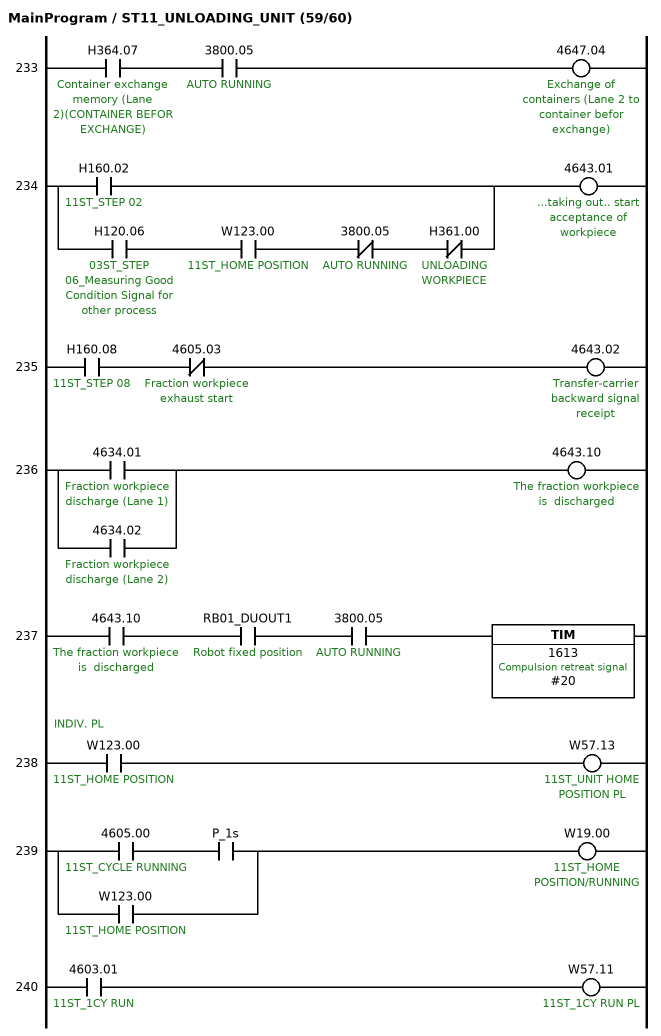
; [picture p576: MainProgram / ST11_UNLOADING_UNIT, rungs 233-240]
; rung 233
LD H364.07  ; Container exchange memory (Lane 2)(CONTAINER BEFOR EXCHANGE)
AND 3800.05  ; AUTO RUNNING
OUT 4647.04  ; Exchange of containers (Lane 2 to container befor exchange)
; rung 234
LD H160.02  ; 11ST_STEP 02
LD H120.06  ; 03ST_STEP 06_Measuring Good Condition Signal for other process
AND W123.00  ; 11ST_HOME POSITION
ANDNOT 3800.05  ; AUTO RUNNING
ANDNOT H361.00  ; UNLOADING WORKPIECE
ORLD
OUT 4643.01  ; ...taking out.. start acceptance of workpiece
; rung 235
LD H160.08  ; 11ST_STEP 08
ANDNOT 4605.03  ; Fraction workpiece exhaust start
OUT 4643.02  ; Transfer-carrier backward signal receipt
; rung 236
LD 4634.01  ; Fraction workpiece discharge (Lane 1)
OR 4634.02  ; Fraction workpiece discharge (Lane 2)
OUT 4643.10  ; The fraction workpiece is  discharged
; rung 237
LD 4643.10  ; The fraction workpiece is  discharged
AND RB01_DUOUT1  ; Robot fixed position
AND 3800.05  ; AUTO RUNNING
TIM 1613 #20  ; Compulsion retreat signal
; rung 238: INDIV. PL
LD W123.00  ; 11ST_HOME POSITION
OUT W57.13  ; 11ST_UNIT HOME POSITION PL
; rung 239
LD 4605.00  ; 11ST_CYCLE RUNNING
AND P_1s
OR W123.00  ; 11ST_HOME POSITION
OUT W19.00  ; 11ST_HOME POSITION/RUNNING
; rung 240
LD 4603.01  ; 11ST_1CY RUN
OUT W57.11  ; 11ST_1CY RUN PL

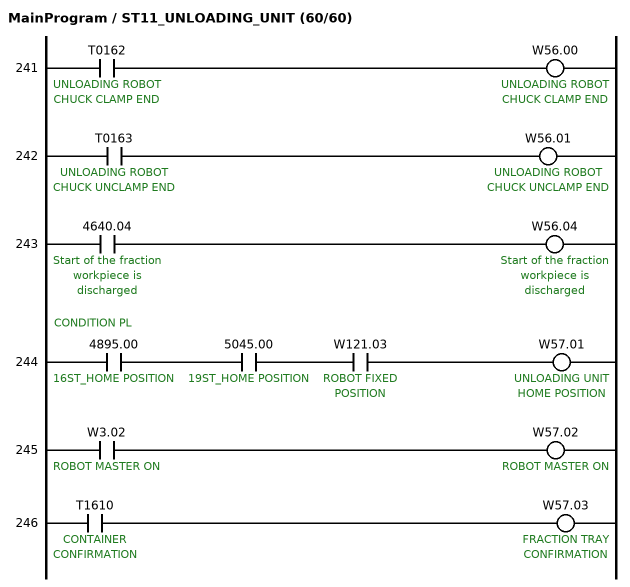
; rung 241
LD T0162  ; UNLOADING ROBOT CHUCK CLAMP END
OUT W56.00  ; UNLOADING ROBOT CHUCK CLAMP END
; rung 242
LD T0163  ; UNLOADING ROBOT CHUCK UNCLAMP END
OUT W56.01  ; UNLOADING ROBOT CHUCK UNCLAMP END
; rung 243
LD 4640.04  ; Start of the fraction workpiece is discharged
OUT W56.04  ; Start of the fraction workpiece is discharged
; rung 244: CONDITION PL
LD 4895.00  ; 16ST_HOME POSITION
AND 5045.00  ; 19ST_HOME POSITION
AND W121.03  ; ROBOT FIXED POSITION
OUT W57.01  ; UNLOADING UNIT HOME POSITION
; rung 245
LD W3.02  ; ROBOT MASTER ON
OUT W57.02  ; ROBOT MASTER ON
; rung 246
LD T1610  ; CONTAINER CONFIRMATION
OUT W57.03  ; FRACTION TRAY CONFIRMATION

### Section ST12_BEARING_SUPPLY_UNIT
; rung 0: 12ST_BEARING SUPPLY UNIT

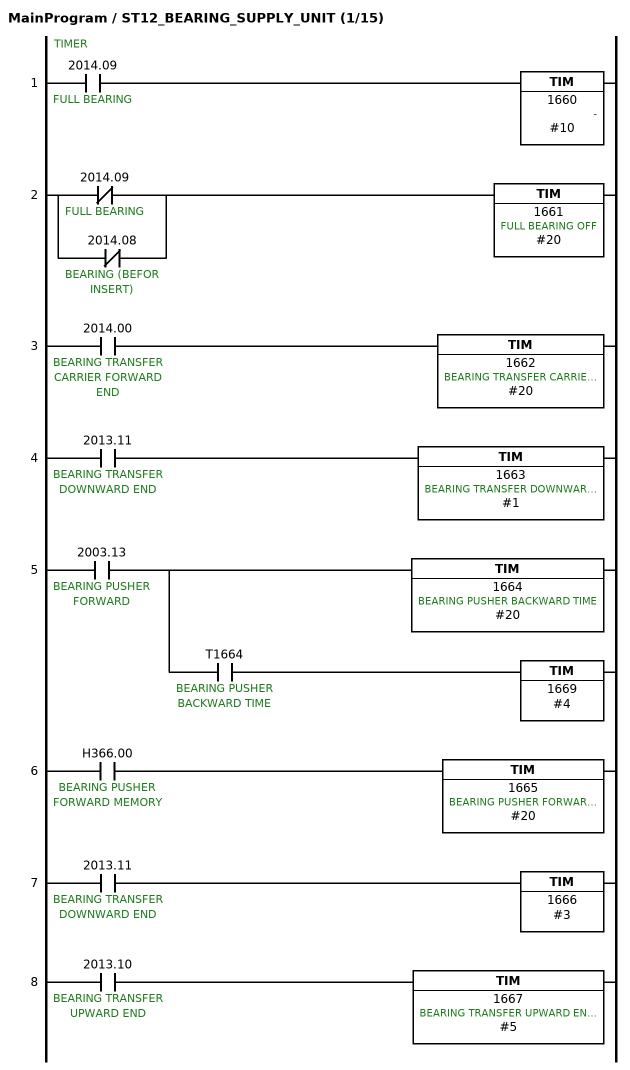
; rung 1: TIMER
LD 2014.09  ; FULL BEARING
TIM 1660 #10  ; -
; rung 2
LDNOT 2014.09  ; FULL BEARING
ORNOT 2014.08  ; BEARING (BEFOR INSERT)
TIM 1661 #20  ; FULL BEARING OFF
; rung 3
LD 2014.00  ; BEARING TRANSFER CARRIER FORWARD END
TIM 1662 #20  ; BEARING TRANSFER CARRIER FORWARD END TIME
; rung 4
LD 2013.11  ; BEARING TRANSFER DOWNWARD END
TIM 1663 #1  ; BEARING TRANSFER DOWNWARD END TIME
; rung 5
LD 2003.13  ; BEARING PUSHER FORWARD
TIM 1664 #20  ; BEARING PUSHER BACKWARD TIME
AND T1664  ; BEARING PUSHER BACKWARD TIME
TIM 1669 #4
; rung 6
LD H366.00  ; BEARING PUSHER FORWARD MEMORY
TIM 1665 #20  ; BEARING PUSHER FORWARD MEMORY TIME
; rung 7
LD 2013.11  ; BEARING TRANSFER DOWNWARD END
TIM 1666 #3
; rung 8
LD 2013.10  ; BEARING TRANSFER UPWARD END
TIM 1667 #5  ; BEARING TRANSFER UPWARD END CONFIRMATION

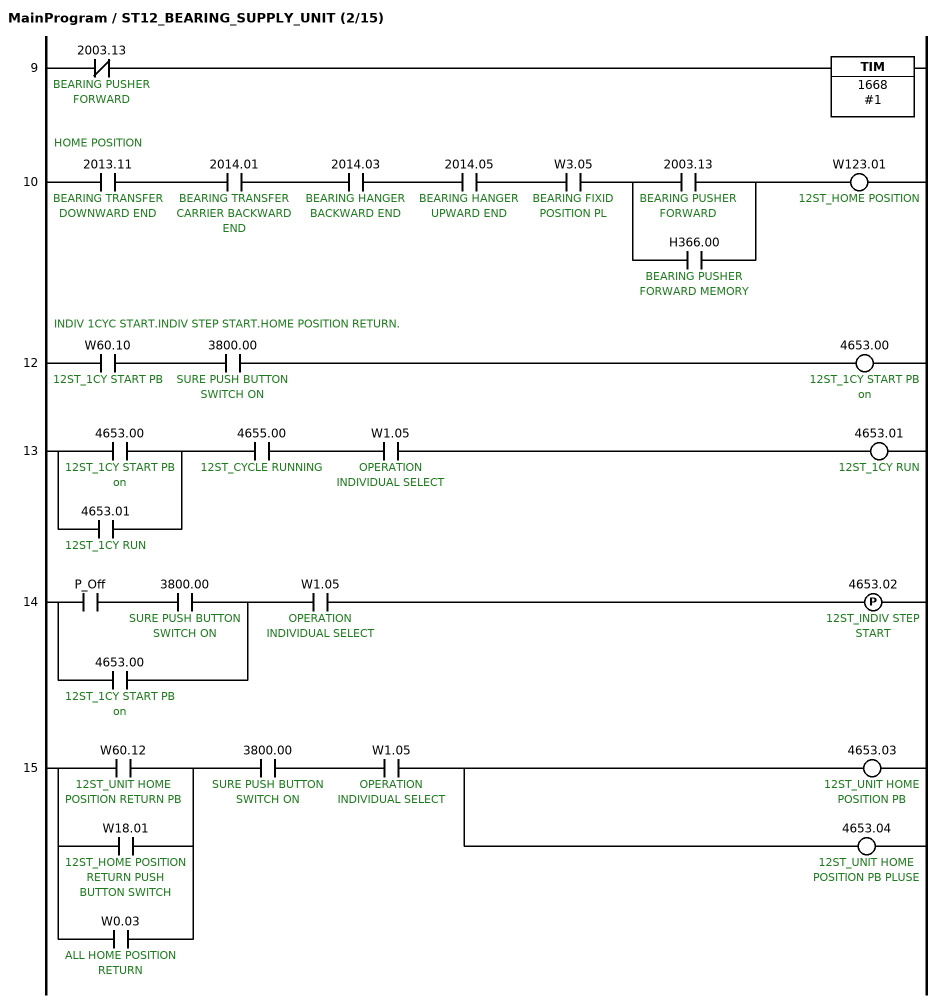
; rung 9
LDNOT 2003.13  ; BEARING PUSHER FORWARD
TIM 1668 #1
; rung 10: HOME POSITION
LD 2013.11  ; BEARING TRANSFER DOWNWARD END
AND 2014.01  ; BEARING TRANSFER CARRIER BACKWARD END
AND 2014.03  ; BEARING HANGER BACKWARD END
AND 2014.05  ; BEARING HANGER UPWARD END
AND W3.05  ; BEARING FIXID POSITION PL
LD 2003.13  ; BEARING PUSHER FORWARD
OR H366.00  ; BEARING PUSHER FORWARD MEMORY
ANDLD
OUT W123.01  ; 12ST_HOME POSITION
; rung 11: INTERFERENCE
; rung 12: INDIV 1CYC START.INDIV STEP START.HOME POSITION RETURN.
LD W60.10  ; 12ST_1CY START PB
AND 3800.00  ; SURE PUSH BUTTON SWITCH ON
OUT 4653.00  ; 12ST_1CY START PB on
; rung 13
LD 4653.00  ; 12ST_1CY START PB on
OR 4653.01  ; 12ST_1CY RUN
AND 4655.00  ; 12ST_CYCLE RUNNING
AND W1.05  ; OPERATION INDIVIDUAL SELECT
OUT 4653.01  ; 12ST_1CY RUN
; rung 14
LD P_Off
AND 3800.00  ; SURE PUSH BUTTON SWITCH ON
OR 4653.00  ; 12ST_1CY START PB on
AND W1.05  ; OPERATION INDIVIDUAL SELECT
DIFU(013) 4653.02  ; 12ST_INDIV STEP START
; rung 15
LD W60.12  ; 12ST_UNIT HOME POSITION RETURN PB
OR W18.01  ; 12ST_HOME POSITION RETURN PUSH BUTTON SWITCH
OR W0.03  ; ALL HOME POSITION RETURN
AND 3800.00  ; SURE PUSH BUTTON SWITCH ON
AND W1.05  ; OPERATION INDIVIDUAL SELECT
OUT 4653.03  ; 12ST_UNIT HOME POSITION PB
OUT 4653.04  ; 12ST_UNIT HOME POSITION PB PLUSE

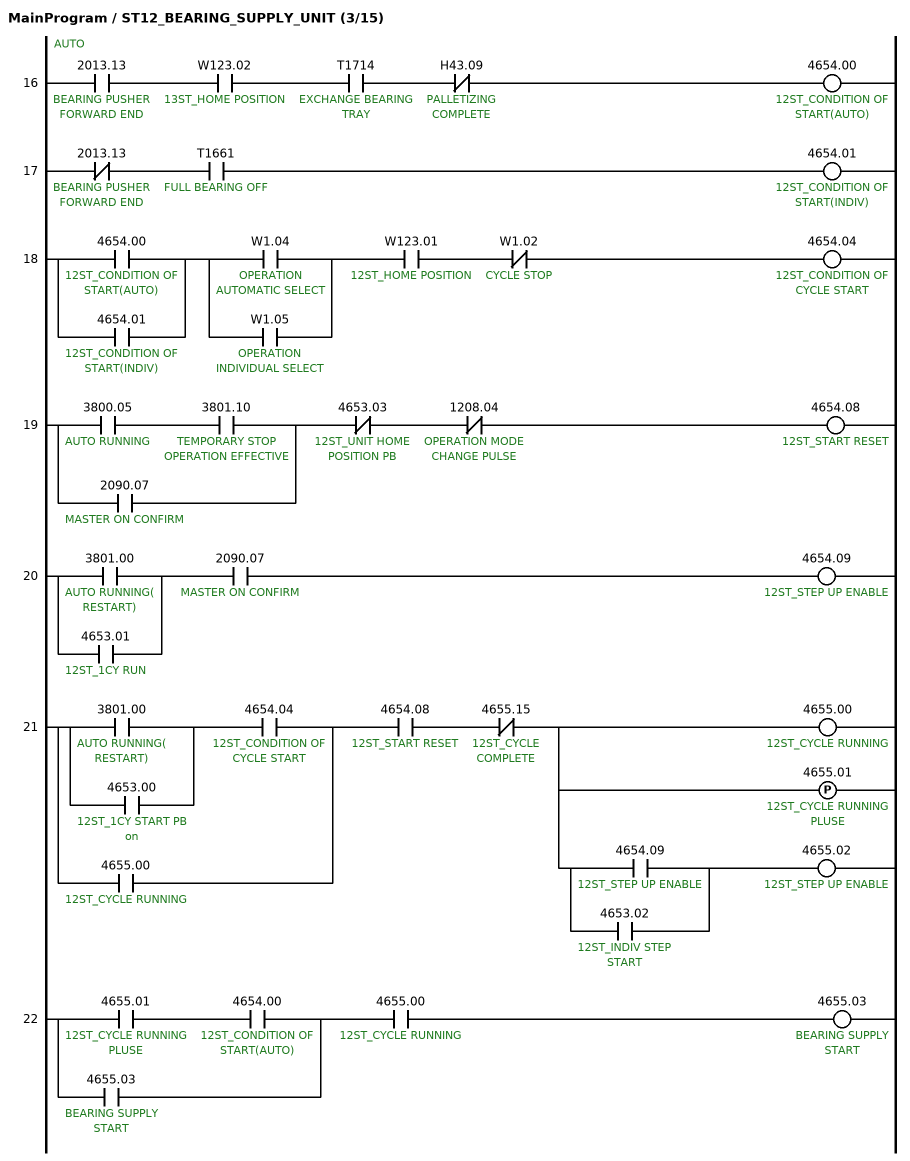
; rung 16: AUTO
LD 2013.13  ; BEARING PUSHER FORWARD END
AND W123.02  ; 13ST_HOME POSITION
AND T1714  ; EXCHANGE BEARING TRAY
ANDNOT H43.09  ; PALLETIZING COMPLETE
OUT 4654.00  ; 12ST_CONDITION OF START(AUTO)
; rung 17
LDNOT 2013.13  ; BEARING PUSHER FORWARD END
AND T1661  ; FULL BEARING OFF
OUT 4654.01  ; 12ST_CONDITION OF START(INDIV)
; rung 18
LD 4654.00  ; 12ST_CONDITION OF START(AUTO)
OR 4654.01  ; 12ST_CONDITION OF START(INDIV)
LD W1.04  ; OPERATION AUTOMATIC SELECT
OR W1.05  ; OPERATION INDIVIDUAL SELECT
ANDLD
AND W123.01  ; 12ST_HOME POSITION
ANDNOT W1.02  ; CYCLE STOP
OUT 4654.04  ; 12ST_CONDITION OF CYCLE START
; rung 19
LD 3800.05  ; AUTO RUNNING
AND 3801.10  ; TEMPORARY STOP OPERATION EFFECTIVE
OR 2090.07  ; MASTER ON CONFIRM
ANDNOT 4653.03  ; 12ST_UNIT HOME POSITION PB
ANDNOT 1208.04  ; OPERATION MODE CHANGE PULSE
OUT 4654.08  ; 12ST_START RESET
; rung 20
LD 3801.00  ; AUTO RUNNING(RESTART)
OR 4653.01  ; 12ST_1CY RUN
AND 2090.07  ; MASTER ON CONFIRM
OUT 4654.09  ; 12ST_STEP UP ENABLE
; rung 21
LD 3801.00  ; AUTO RUNNING(RESTART)
OR 4653.00  ; 12ST_1CY START PB on
AND 4654.04  ; 12ST_CONDITION OF CYCLE START
OR 4655.00  ; 12ST_CYCLE RUNNING
AND 4654.08  ; 12ST_START RESET
ANDNOT 4655.15  ; 12ST_CYCLE COMPLETE
OUT 4655.00  ; 12ST_CYCLE RUNNING
DIFU(013) 4655.01  ; 12ST_CYCLE RUNNING PLUSE
LD 4654.09  ; 12ST_STEP UP ENABLE
OR 4653.02  ; 12ST_INDIV STEP START
ANDLD
OUT 4655.02  ; 12ST_STEP UP ENABLE
; rung 22
LD 4655.01  ; 12ST_CYCLE RUNNING PLUSE
AND 4654.00  ; 12ST_CONDITION OF START(AUTO)
OR 4655.03  ; BEARING SUPPLY START
AND 4655.00  ; 12ST_CYCLE RUNNING
OUT 4655.03  ; BEARING SUPPLY START

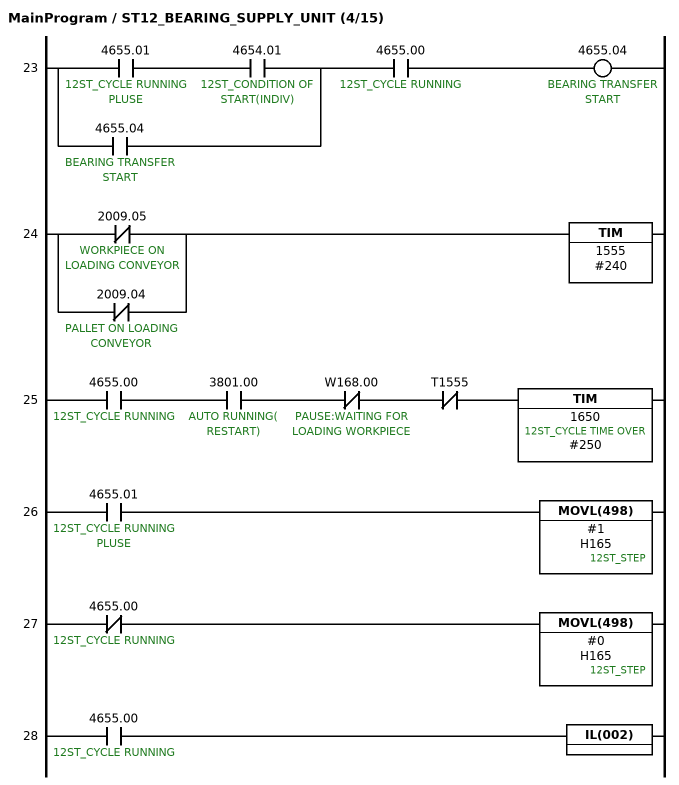
; rung 23
LD 4655.01  ; 12ST_CYCLE RUNNING PLUSE
AND 4654.01  ; 12ST_CONDITION OF START(INDIV)
OR 4655.04  ; BEARING TRANSFER START
AND 4655.00  ; 12ST_CYCLE RUNNING
OUT 4655.04  ; BEARING TRANSFER START
; rung 24
LDNOT 2009.05  ; WORKPIECE ON LOADING CONVEYOR
ORNOT 2009.04  ; PALLET ON LOADING CONVEYOR
TIM 1555 #240
; rung 25
LD 4655.00  ; 12ST_CYCLE RUNNING
AND 3801.00  ; AUTO RUNNING(RESTART)
ANDNOT W168.00  ; PAUSE:WAITING FOR LOADING WORKPIECE
ANDNOT T1555
TIM 1650 #250  ; 12ST_CYCLE TIME OVER
; rung 26
LD 4655.01  ; 12ST_CYCLE RUNNING PLUSE
MOVL(498) #1 H165  ; 12ST_STEP
; rung 27
LDNOT 4655.00  ; 12ST_CYCLE RUNNING
MOVL(498) #0 H165  ; 12ST_STEP
; rung 28
LD 4655.00  ; 12ST_CYCLE RUNNING
IL(002)

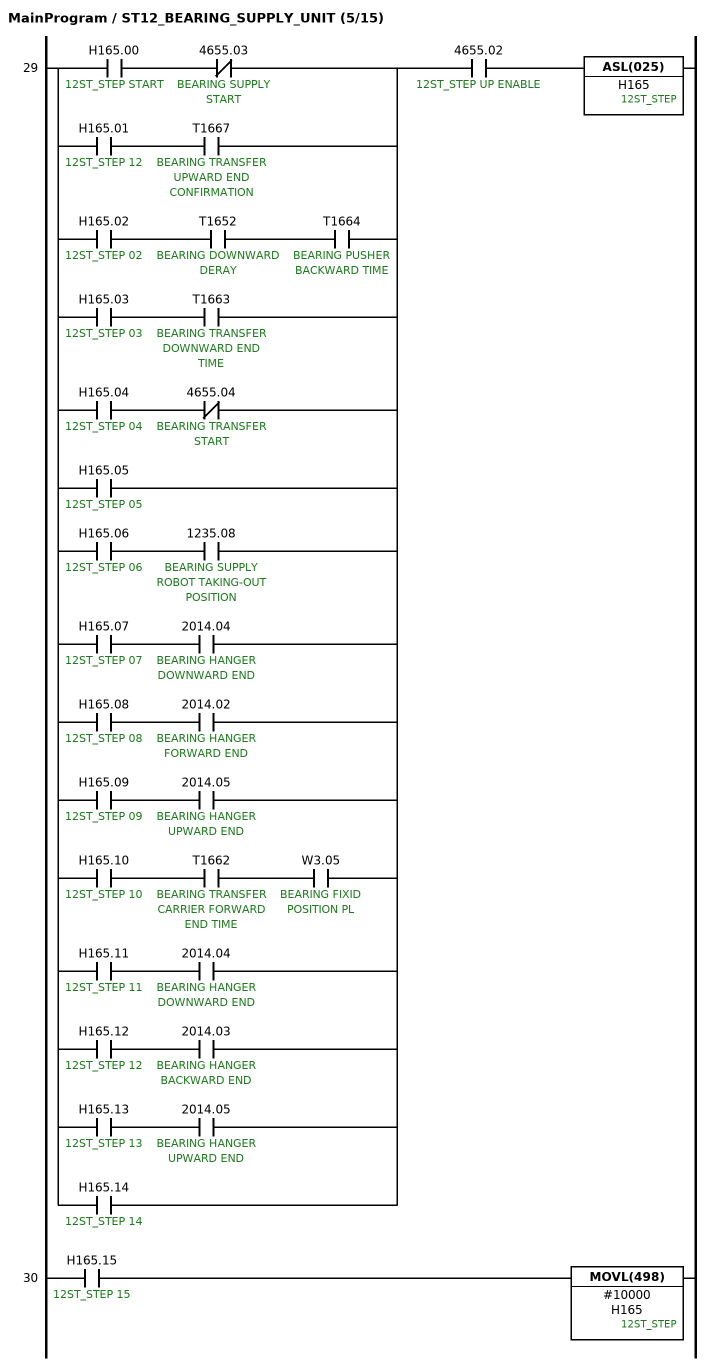
; rung 29
LD H165.00  ; 12ST_STEP START
ANDNOT 4655.03  ; BEARING SUPPLY START
LD H165.01  ; 12ST_STEP 12
AND T1667  ; BEARING TRANSFER UPWARD END CONFIRMATION
ORLD
LD H165.02  ; 12ST_STEP 02
AND T1652  ; BEARING DOWNWARD DERAY
AND T1664  ; BEARING PUSHER BACKWARD TIME
ORLD
LD H165.03  ; 12ST_STEP 03
AND T1663  ; BEARING TRANSFER DOWNWARD END TIME
ORLD
LD H165.04  ; 12ST_STEP 04
ANDNOT 4655.04  ; BEARING TRANSFER START
ORLD
OR H165.05  ; 12ST_STEP 05
LD H165.06  ; 12ST_STEP 06
AND 1235.08  ; BEARING SUPPLY ROBOT TAKING-OUT POSITION
ORLD
LD H165.07  ; 12ST_STEP 07
AND 2014.04  ; BEARING HANGER DOWNWARD END
ORLD
LD H165.08  ; 12ST_STEP 08
AND 2014.02  ; BEARING HANGER FORWARD END
ORLD
LD H165.09  ; 12ST_STEP 09
AND 2014.05  ; BEARING HANGER UPWARD END
ORLD
LD H165.10  ; 12ST_STEP 10
AND T1662  ; BEARING TRANSFER CARRIER FORWARD END TIME
AND W3.05  ; BEARING FIXID POSITION PL
ORLD
LD H165.11  ; 12ST_STEP 11
AND 2014.04  ; BEARING HANGER DOWNWARD END
ORLD
LD H165.12  ; 12ST_STEP 12
AND 2014.03  ; BEARING HANGER BACKWARD END
ORLD
LD H165.13  ; 12ST_STEP 13
AND 2014.05  ; BEARING HANGER UPWARD END
ORLD
OR H165.14  ; 12ST_STEP 14
AND 4655.02  ; 12ST_STEP UP ENABLE
ASL(025) H165  ; 12ST_STEP
; rung 30
LD H165.15  ; 12ST_STEP 15
MOVL(498) #10000 H165  ; 12ST_STEP

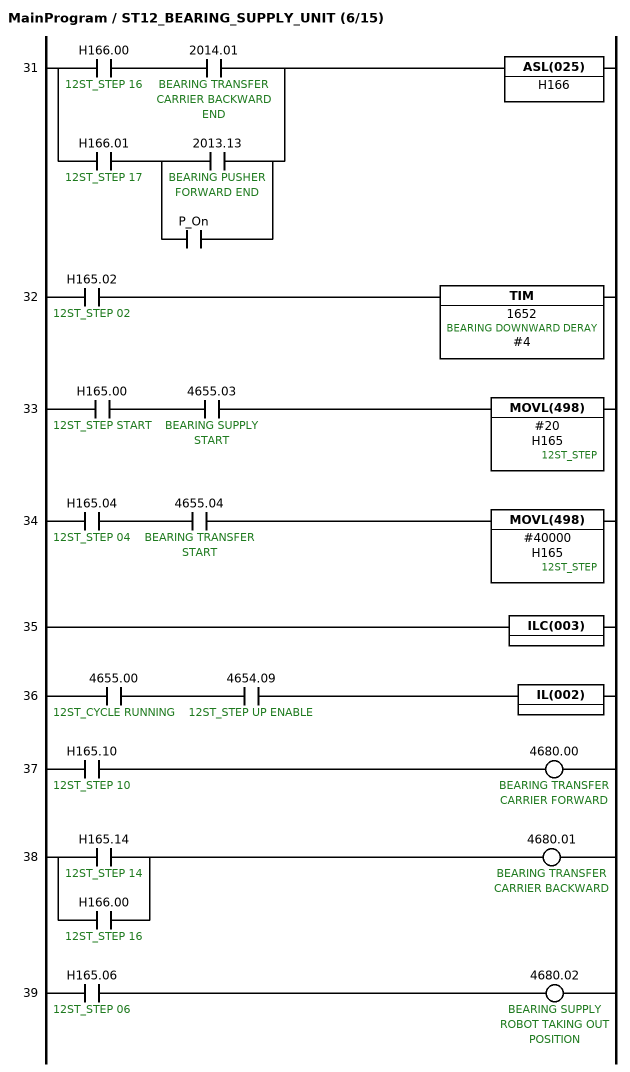
; rung 31
LD H166.00  ; 12ST_STEP 16
AND 2014.01  ; BEARING TRANSFER CARRIER BACKWARD END
LD H166.01  ; 12ST_STEP 17
LD 2013.13  ; BEARING PUSHER FORWARD END
OR P_On
ANDLD
ORLD
ASL(025) H166
; rung 32
LD H165.02  ; 12ST_STEP 02
TIM 1652 #4  ; BEARING DOWNWARD DERAY
; rung 33
LD H165.00  ; 12ST_STEP START
AND 4655.03  ; BEARING SUPPLY START
MOVL(498) #20 H165  ; 12ST_STEP
; rung 34
LD H165.04  ; 12ST_STEP 04
AND 4655.04  ; BEARING TRANSFER START
MOVL(498) #40000 H165  ; 12ST_STEP
; rung 35
ILC(003)
; rung 36
LD 4655.00  ; 12ST_CYCLE RUNNING
AND 4654.09  ; 12ST_STEP UP ENABLE
IL(002)
; rung 37
LD H165.10  ; 12ST_STEP 10
OUT 4680.00  ; BEARING TRANSFER CARRIER FORWARD
; rung 38
LD H165.14  ; 12ST_STEP 14
OR H166.00  ; 12ST_STEP 16
OUT 4680.01  ; BEARING TRANSFER CARRIER BACKWARD
; rung 39
LD H165.06  ; 12ST_STEP 06
OUT 4680.02  ; BEARING SUPPLY ROBOT TAKING OUT POSITION

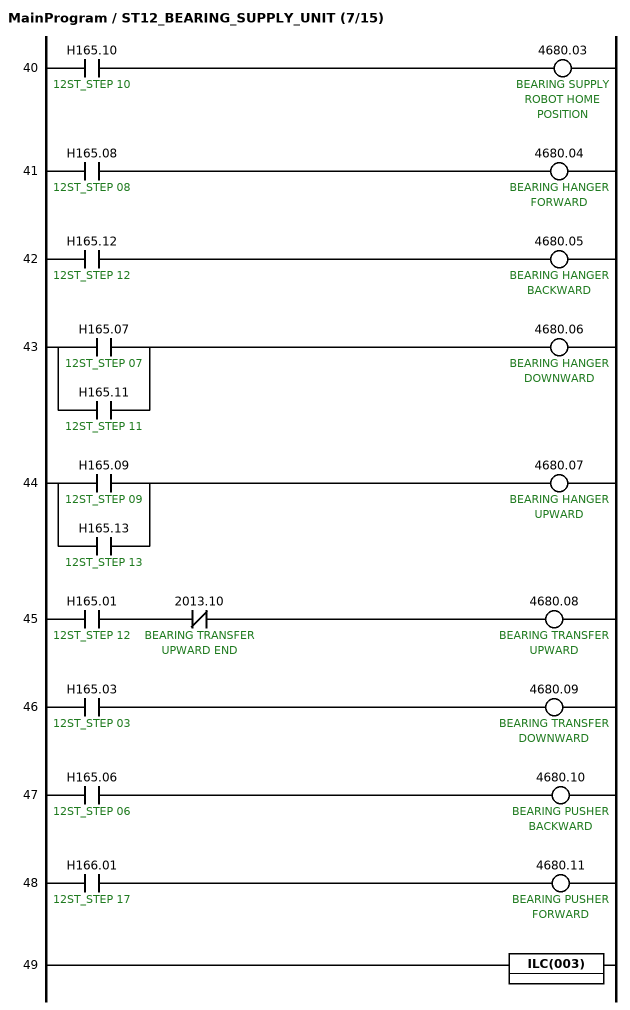
; rung 40
LD H165.10  ; 12ST_STEP 10
OUT 4680.03  ; BEARING SUPPLY ROBOT HOME POSITION
; rung 41
LD H165.08  ; 12ST_STEP 08
OUT 4680.04  ; BEARING HANGER FORWARD
; rung 42
LD H165.12  ; 12ST_STEP 12
OUT 4680.05  ; BEARING HANGER BACKWARD
; rung 43
LD H165.07  ; 12ST_STEP 07
OR H165.11  ; 12ST_STEP 11
OUT 4680.06  ; BEARING HANGER DOWNWARD
; rung 44
LD H165.09  ; 12ST_STEP 09
OR H165.13  ; 12ST_STEP 13
OUT 4680.07  ; BEARING HANGER UPWARD
; rung 45
LD H165.01  ; 12ST_STEP 12
ANDNOT 2013.10  ; BEARING TRANSFER UPWARD END
OUT 4680.08  ; BEARING TRANSFER UPWARD
; rung 46
LD H165.03  ; 12ST_STEP 03
OUT 4680.09  ; BEARING TRANSFER DOWNWARD
; rung 47
LD H165.06  ; 12ST_STEP 06
OUT 4680.10  ; BEARING PUSHER BACKWARD
; rung 48
LD H166.01  ; 12ST_STEP 17
OUT 4680.11  ; BEARING PUSHER FORWARD
; rung 49
ILC(003)

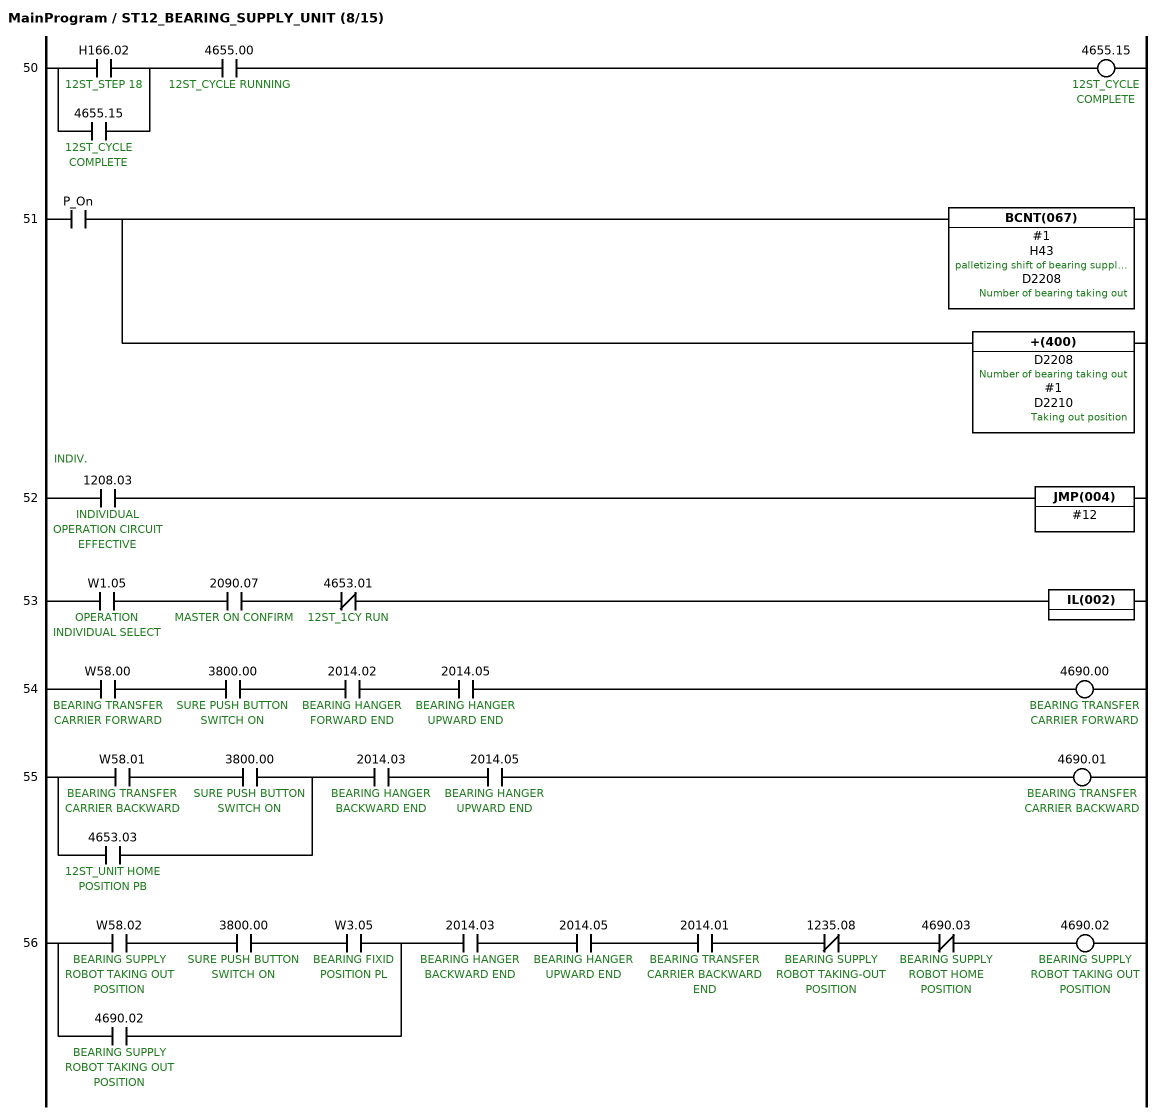
; rung 50
LD H166.02  ; 12ST_STEP 18
OR 4655.15  ; 12ST_CYCLE COMPLETE
AND 4655.00  ; 12ST_CYCLE RUNNING
OUT 4655.15  ; 12ST_CYCLE COMPLETE
; rung 51
LD P_On
BCNT(067) #1 H43 D2208  ; palletizing shift of bearing supply robot, Number of bearing taking out
+(400) D2208 #1 D2210  ; Number of bearing taking out, Taking out position
; rung 52: INDIV.
LD 1208.03  ; INDIVIDUAL OPERATION CIRCUIT EFFECTIVE
JMP(004) #12
; rung 53
LD W1.05  ; OPERATION INDIVIDUAL SELECT
AND 2090.07  ; MASTER ON CONFIRM
ANDNOT 4653.01  ; 12ST_1CY RUN
IL(002)
; rung 54
LD W58.00  ; BEARING TRANSFER CARRIER FORWARD
AND 3800.00  ; SURE PUSH BUTTON SWITCH ON
AND 2014.02  ; BEARING HANGER FORWARD END
AND 2014.05  ; BEARING HANGER UPWARD END
OUT 4690.00  ; BEARING TRANSFER CARRIER FORWARD
; rung 55
LD W58.01  ; BEARING TRANSFER CARRIER BACKWARD
AND 3800.00  ; SURE PUSH BUTTON SWITCH ON
OR 4653.03  ; 12ST_UNIT HOME POSITION PB
AND 2014.03  ; BEARING HANGER BACKWARD END
AND 2014.05  ; BEARING HANGER UPWARD END
OUT 4690.01  ; BEARING TRANSFER CARRIER BACKWARD
; rung 56
LD W58.02  ; BEARING SUPPLY ROBOT TAKING OUT POSITION
AND 3800.00  ; SURE PUSH BUTTON SWITCH ON
AND W3.05  ; BEARING FIXID POSITION PL
OR 4690.02  ; BEARING SUPPLY ROBOT TAKING OUT POSITION
AND 2014.03  ; BEARING HANGER BACKWARD END
AND 2014.05  ; BEARING HANGER UPWARD END
AND 2014.01  ; BEARING TRANSFER CARRIER BACKWARD END
ANDNOT 1235.08  ; BEARING SUPPLY ROBOT TAKING-OUT POSITION
ANDNOT 4690.03  ; BEARING SUPPLY ROBOT HOME POSITION
OUT 4690.02  ; BEARING SUPPLY ROBOT TAKING OUT POSITION

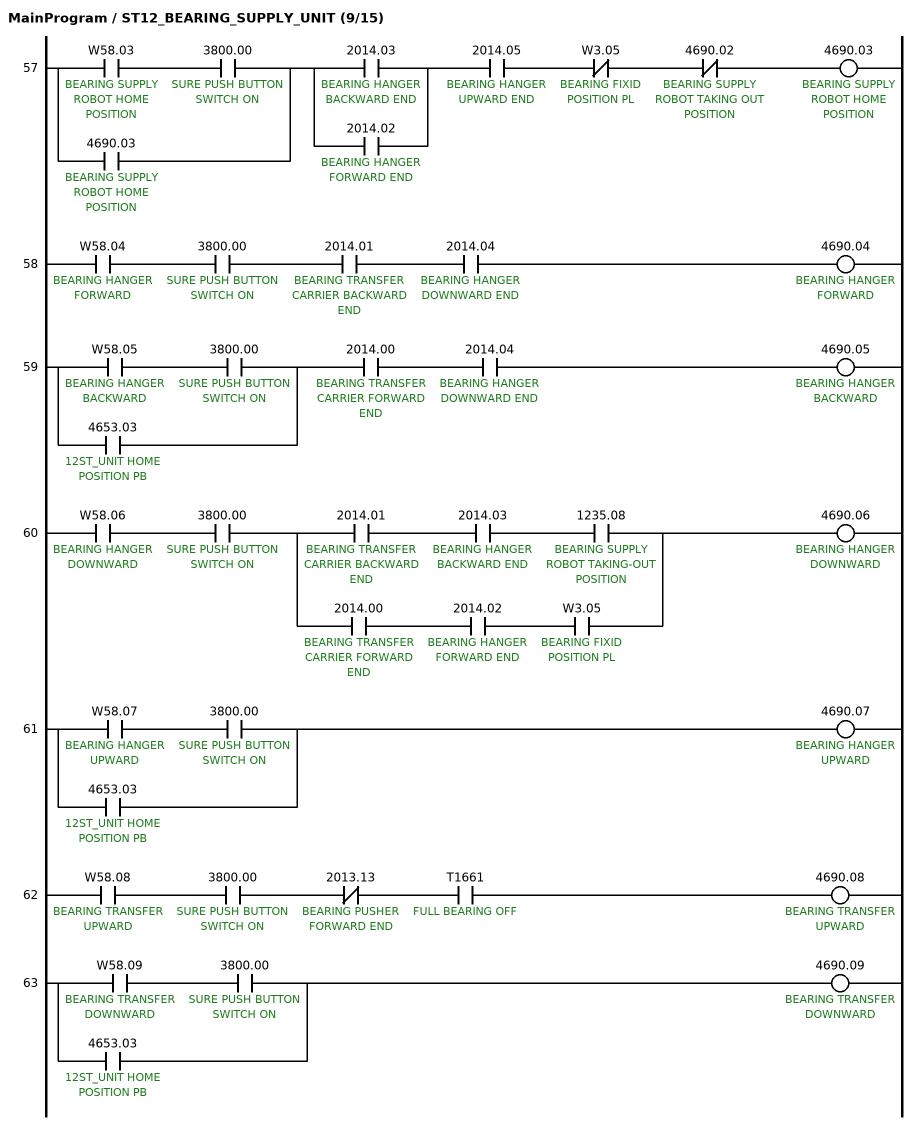
; rung 57
LD W58.03  ; BEARING SUPPLY ROBOT HOME POSITION
AND 3800.00  ; SURE PUSH BUTTON SWITCH ON
OR 4690.03  ; BEARING SUPPLY ROBOT HOME POSITION
LD 2014.03  ; BEARING HANGER BACKWARD END
OR 2014.02  ; BEARING HANGER FORWARD END
ANDLD
AND 2014.05  ; BEARING HANGER UPWARD END
ANDNOT W3.05  ; BEARING FIXID POSITION PL
ANDNOT 4690.02  ; BEARING SUPPLY ROBOT TAKING OUT POSITION
OUT 4690.03  ; BEARING SUPPLY ROBOT HOME POSITION
; rung 58
LD W58.04  ; BEARING HANGER FORWARD
AND 3800.00  ; SURE PUSH BUTTON SWITCH ON
AND 2014.01  ; BEARING TRANSFER CARRIER BACKWARD END
AND 2014.04  ; BEARING HANGER DOWNWARD END
OUT 4690.04  ; BEARING HANGER FORWARD
; rung 59
LD W58.05  ; BEARING HANGER BACKWARD
AND 3800.00  ; SURE PUSH BUTTON SWITCH ON
OR 4653.03  ; 12ST_UNIT HOME POSITION PB
AND 2014.00  ; BEARING TRANSFER CARRIER FORWARD END
AND 2014.04  ; BEARING HANGER DOWNWARD END
OUT 4690.05  ; BEARING HANGER BACKWARD
; rung 60
LD W58.06  ; BEARING HANGER DOWNWARD
AND 3800.00  ; SURE PUSH BUTTON SWITCH ON
LD 2014.01  ; BEARING TRANSFER CARRIER BACKWARD END
AND 2014.03  ; BEARING HANGER BACKWARD END
AND 1235.08  ; BEARING SUPPLY ROBOT TAKING-OUT POSITION
LD 2014.00  ; BEARING TRANSFER CARRIER FORWARD END
AND 2014.02  ; BEARING HANGER FORWARD END
AND W3.05  ; BEARING FIXID POSITION PL
ORLD
ANDLD
OUT 4690.06  ; BEARING HANGER DOWNWARD
; rung 61
LD W58.07  ; BEARING HANGER UPWARD
AND 3800.00  ; SURE PUSH BUTTON SWITCH ON
OR 4653.03  ; 12ST_UNIT HOME POSITION PB
OUT 4690.07  ; BEARING HANGER UPWARD
; rung 62
LD W58.08  ; BEARING TRANSFER UPWARD
AND 3800.00  ; SURE PUSH BUTTON SWITCH ON
ANDNOT 2013.13  ; BEARING PUSHER FORWARD END
AND T1661  ; FULL BEARING OFF
OUT 4690.08  ; BEARING TRANSFER UPWARD
; rung 63
LD W58.09  ; BEARING TRANSFER DOWNWARD
AND 3800.00  ; SURE PUSH BUTTON SWITCH ON
OR 4653.03  ; 12ST_UNIT HOME POSITION PB
OUT 4690.09  ; BEARING TRANSFER DOWNWARD

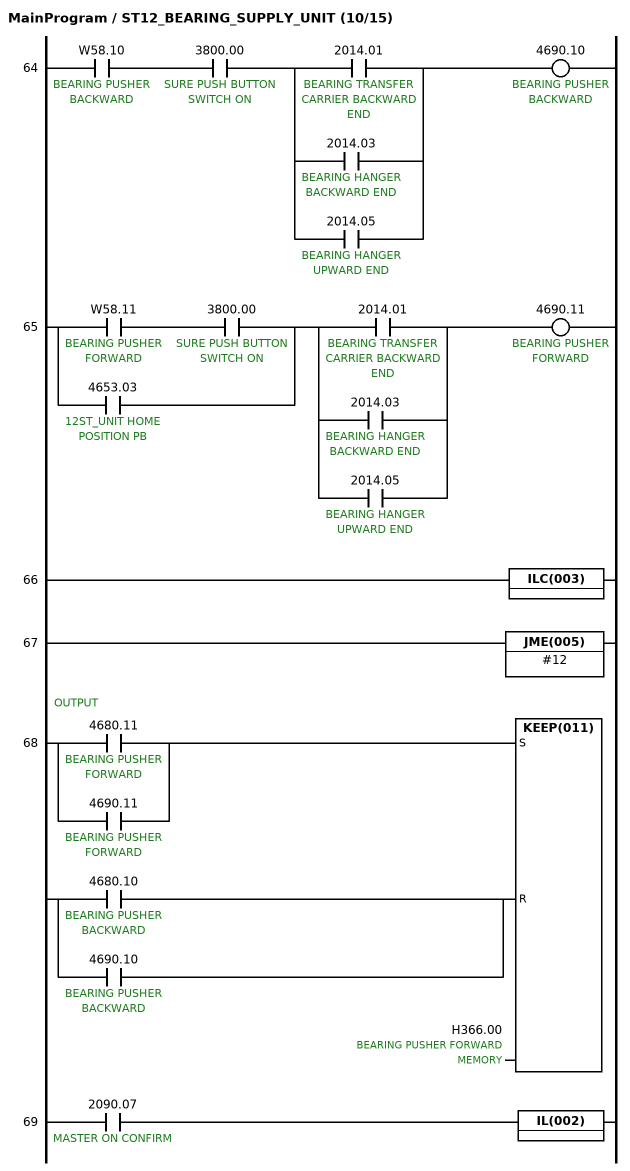
; rung 64
LD W58.10  ; BEARING PUSHER BACKWARD
AND 3800.00  ; SURE PUSH BUTTON SWITCH ON
LD 2014.01  ; BEARING TRANSFER CARRIER BACKWARD END
OR 2014.03  ; BEARING HANGER BACKWARD END
OR 2014.05  ; BEARING HANGER UPWARD END
ANDLD
OUT 4690.10  ; BEARING PUSHER BACKWARD
; rung 65
LD W58.11  ; BEARING PUSHER FORWARD
AND 3800.00  ; SURE PUSH BUTTON SWITCH ON
OR 4653.03  ; 12ST_UNIT HOME POSITION PB
LD 2014.01  ; BEARING TRANSFER CARRIER BACKWARD END
OR 2014.03  ; BEARING HANGER BACKWARD END
OR 2014.05  ; BEARING HANGER UPWARD END
ANDLD
OUT 4690.11  ; BEARING PUSHER FORWARD
; rung 66
ILC(003)
; rung 67
JME(005) #12
; rung 68: OUTPUT
LD 4680.11  ; BEARING PUSHER FORWARD
OR 4690.11  ; BEARING PUSHER FORWARD
LD 4680.10  ; BEARING PUSHER BACKWARD
OR 4690.10  ; BEARING PUSHER BACKWARD
KEEP(011) H366.00  ; BEARING PUSHER FORWARD MEMORY
; rung 69
LD 2090.07  ; MASTER ON CONFIRM
IL(002)

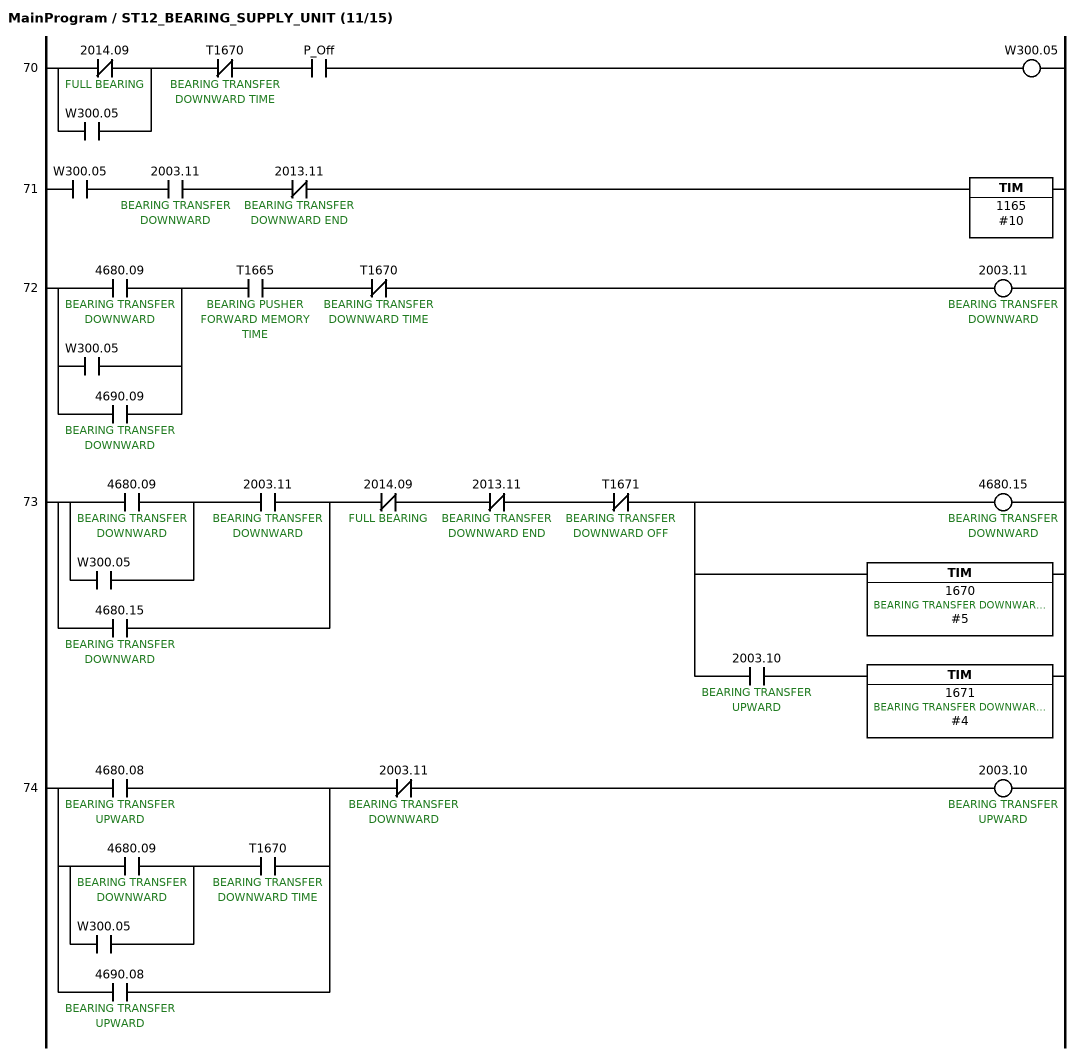
; rung 70
LDNOT 2014.09  ; FULL BEARING
OR W300.05
ANDNOT T1670  ; BEARING TRANSFER DOWNWARD TIME
AND P_Off
OUT W300.05
; rung 71
LD W300.05
AND 2003.11  ; BEARING TRANSFER DOWNWARD
ANDNOT 2013.11  ; BEARING TRANSFER DOWNWARD END
TIM 1165 #10
; rung 72
LD 4680.09  ; BEARING TRANSFER DOWNWARD
OR W300.05
OR 4690.09  ; BEARING TRANSFER DOWNWARD
AND T1665  ; BEARING PUSHER FORWARD MEMORY TIME
ANDNOT T1670  ; BEARING TRANSFER DOWNWARD TIME
OUT 2003.11  ; BEARING TRANSFER DOWNWARD
; rung 73
LD 4680.09  ; BEARING TRANSFER DOWNWARD
OR W300.05
AND 2003.11  ; BEARING TRANSFER DOWNWARD
OR 4680.15  ; BEARING TRANSFER DOWNWARD
ANDNOT 2014.09  ; FULL BEARING
ANDNOT 2013.11  ; BEARING TRANSFER DOWNWARD END
ANDNOT T1671  ; BEARING TRANSFER DOWNWARD OFF
OUT 4680.15  ; BEARING TRANSFER DOWNWARD
TIM 1670 #5  ; BEARING TRANSFER DOWNWARD TIME
AND 2003.10  ; BEARING TRANSFER UPWARD
TIM 1671 #4  ; BEARING TRANSFER DOWNWARD OFF
; rung 74
LD 4680.08  ; BEARING TRANSFER UPWARD
LD 4680.09  ; BEARING TRANSFER DOWNWARD
OR W300.05
AND T1670  ; BEARING TRANSFER DOWNWARD TIME
ORLD
OR 4690.08  ; BEARING TRANSFER UPWARD
ANDNOT 2003.11  ; BEARING TRANSFER DOWNWARD
OUT 2003.10  ; BEARING TRANSFER UPWARD

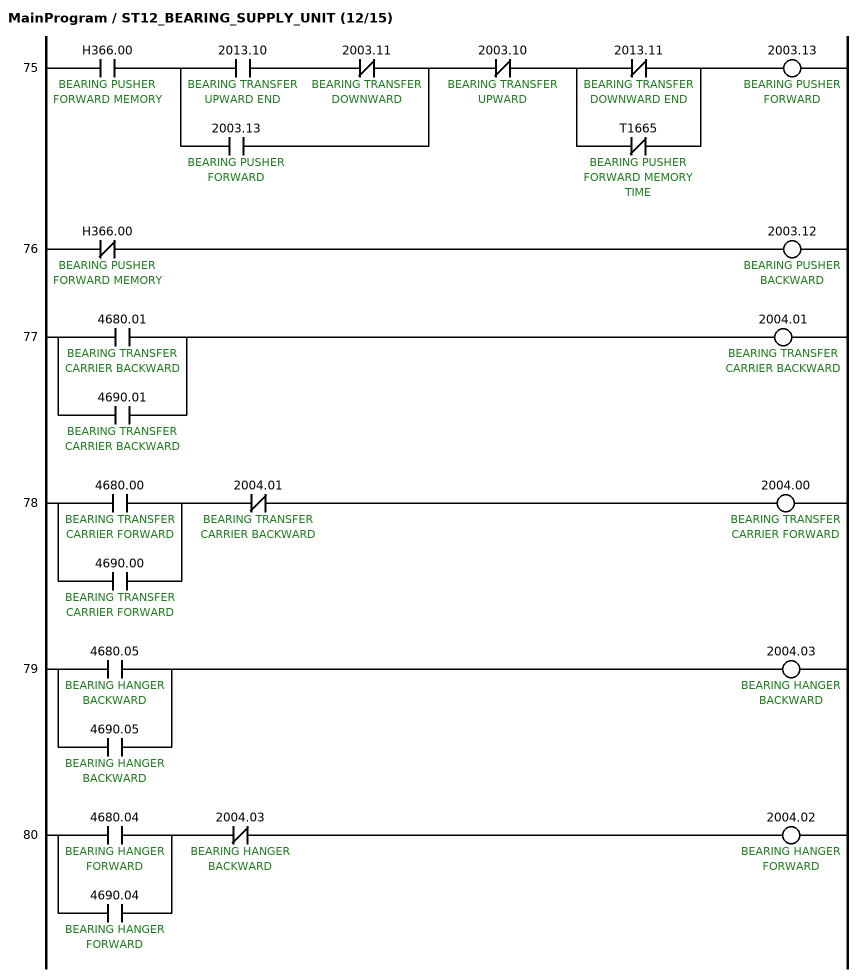
; rung 75
LD H366.00  ; BEARING PUSHER FORWARD MEMORY
LD 2013.10  ; BEARING TRANSFER UPWARD END
ANDNOT 2003.11  ; BEARING TRANSFER DOWNWARD
OR 2003.13  ; BEARING PUSHER FORWARD
ANDLD
ANDNOT 2003.10  ; BEARING TRANSFER UPWARD
LDNOT 2013.11  ; BEARING TRANSFER DOWNWARD END
ORNOT T1665  ; BEARING PUSHER FORWARD MEMORY TIME
ANDLD
OUT 2003.13  ; BEARING PUSHER FORWARD
; rung 76
LDNOT H366.00  ; BEARING PUSHER FORWARD MEMORY
OUT 2003.12  ; BEARING PUSHER BACKWARD
; rung 77
LD 4680.01  ; BEARING TRANSFER CARRIER BACKWARD
OR 4690.01  ; BEARING TRANSFER CARRIER BACKWARD
OUT 2004.01  ; BEARING TRANSFER CARRIER BACKWARD
; rung 78
LD 4680.00  ; BEARING TRANSFER CARRIER FORWARD
OR 4690.00  ; BEARING TRANSFER CARRIER FORWARD
ANDNOT 2004.01  ; BEARING TRANSFER CARRIER BACKWARD
OUT 2004.00  ; BEARING TRANSFER CARRIER FORWARD
; rung 79
LD 4680.05  ; BEARING HANGER BACKWARD
OR 4690.05  ; BEARING HANGER BACKWARD
OUT 2004.03  ; BEARING HANGER BACKWARD
; rung 80
LD 4680.04  ; BEARING HANGER FORWARD
OR 4690.04  ; BEARING HANGER FORWARD
ANDNOT 2004.03  ; BEARING HANGER BACKWARD
OUT 2004.02  ; BEARING HANGER FORWARD

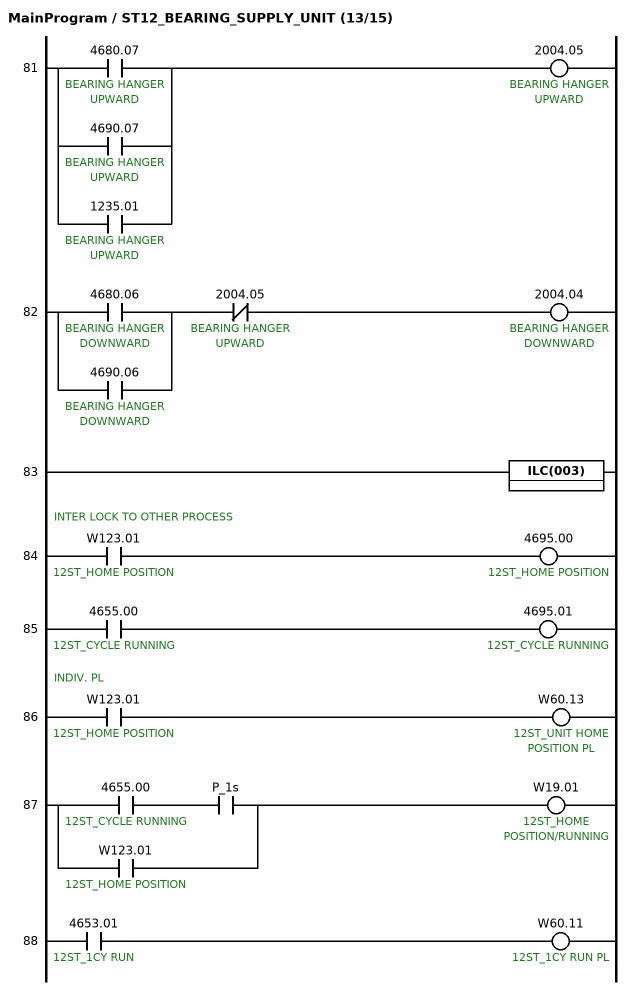
; rung 81
LD 4680.07  ; BEARING HANGER UPWARD
OR 4690.07  ; BEARING HANGER UPWARD
OR 1235.01  ; BEARING HANGER UPWARD
OUT 2004.05  ; BEARING HANGER UPWARD
; rung 82
LD 4680.06  ; BEARING HANGER DOWNWARD
OR 4690.06  ; BEARING HANGER DOWNWARD
ANDNOT 2004.05  ; BEARING HANGER UPWARD
OUT 2004.04  ; BEARING HANGER DOWNWARD
; rung 83
ILC(003)
; rung 84: INTER LOCK TO OTHER PROCESS
LD W123.01  ; 12ST_HOME POSITION
OUT 4695.00  ; 12ST_HOME POSITION
; rung 85
LD 4655.00  ; 12ST_CYCLE RUNNING
OUT 4695.01  ; 12ST_CYCLE RUNNING
; rung 86: INDIV. PL
LD W123.01  ; 12ST_HOME POSITION
OUT W60.13  ; 12ST_UNIT HOME POSITION PL
; rung 87
LD 4655.00  ; 12ST_CYCLE RUNNING
AND P_1s
OR W123.01  ; 12ST_HOME POSITION
OUT W19.01  ; 12ST_HOME POSITION/RUNNING
; rung 88
LD 4653.01  ; 12ST_1CY RUN
OUT W60.11  ; 12ST_1CY RUN PL

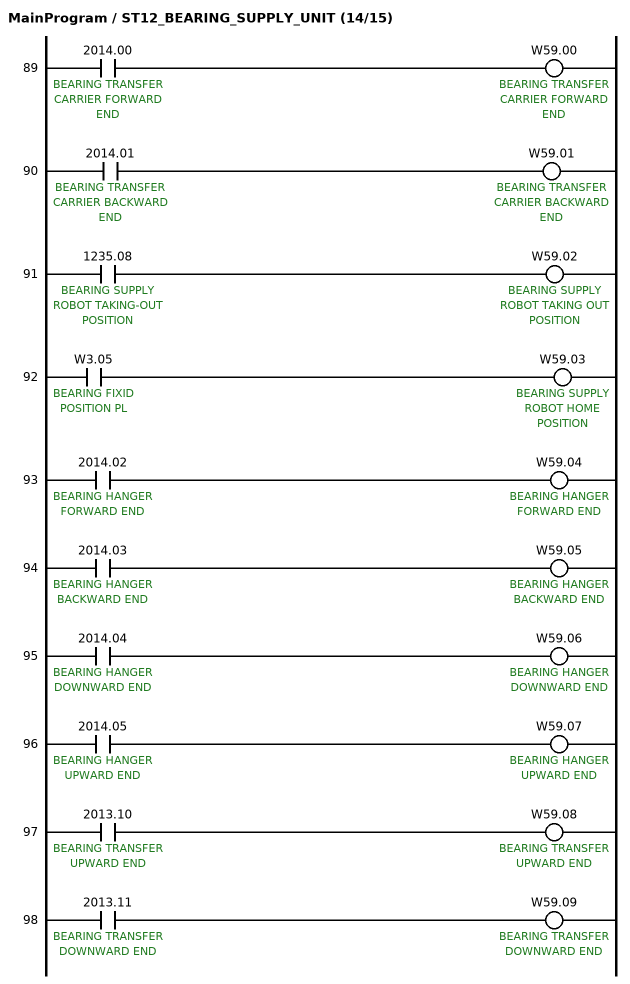
; rung 89
LD 2014.00  ; BEARING TRANSFER CARRIER FORWARD END
OUT W59.00  ; BEARING TRANSFER CARRIER FORWARD END
; rung 90
LD 2014.01  ; BEARING TRANSFER CARRIER BACKWARD END
OUT W59.01  ; BEARING TRANSFER CARRIER BACKWARD END
; rung 91
LD 1235.08  ; BEARING SUPPLY ROBOT TAKING-OUT POSITION
OUT W59.02  ; BEARING SUPPLY ROBOT TAKING OUT POSITION
; rung 92
LD W3.05  ; BEARING FIXID POSITION PL
OUT W59.03  ; BEARING SUPPLY ROBOT HOME POSITION
; rung 93
LD 2014.02  ; BEARING HANGER FORWARD END
OUT W59.04  ; BEARING HANGER FORWARD END
; rung 94
LD 2014.03  ; BEARING HANGER BACKWARD END
OUT W59.05  ; BEARING HANGER BACKWARD END
; rung 95
LD 2014.04  ; BEARING HANGER DOWNWARD END
OUT W59.06  ; BEARING HANGER DOWNWARD END
; rung 96
LD 2014.05  ; BEARING HANGER UPWARD END
OUT W59.07  ; BEARING HANGER UPWARD END
; rung 97
LD 2013.10  ; BEARING TRANSFER UPWARD END
OUT W59.08  ; BEARING TRANSFER UPWARD END
; rung 98
LD 2013.11  ; BEARING TRANSFER DOWNWARD END
OUT W59.09  ; BEARING TRANSFER DOWNWARD END

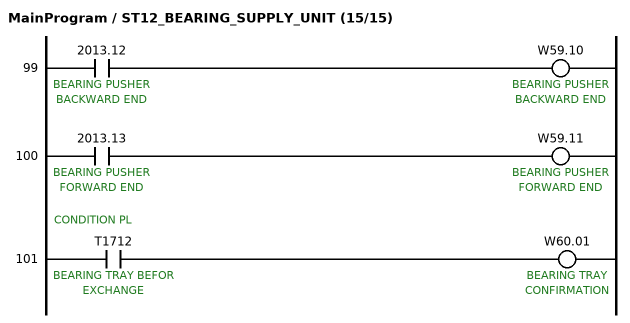
; rung 99
LD 2013.12  ; BEARING PUSHER BACKWARD END
OUT W59.10  ; BEARING PUSHER BACKWARD END
; rung 100
LD 2013.13  ; BEARING PUSHER FORWARD END
OUT W59.11  ; BEARING PUSHER FORWARD END
; rung 101: CONDITION PL
LD T1712  ; BEARING TRAY BEFOR EXCHANGE
OUT W60.01  ; BEARING TRAY CONFIRMATION

### Section ST13_BEARING_EXCHANGE_UNIT
; rung 0: 13ST_BEARING EXCHANGE UNIT

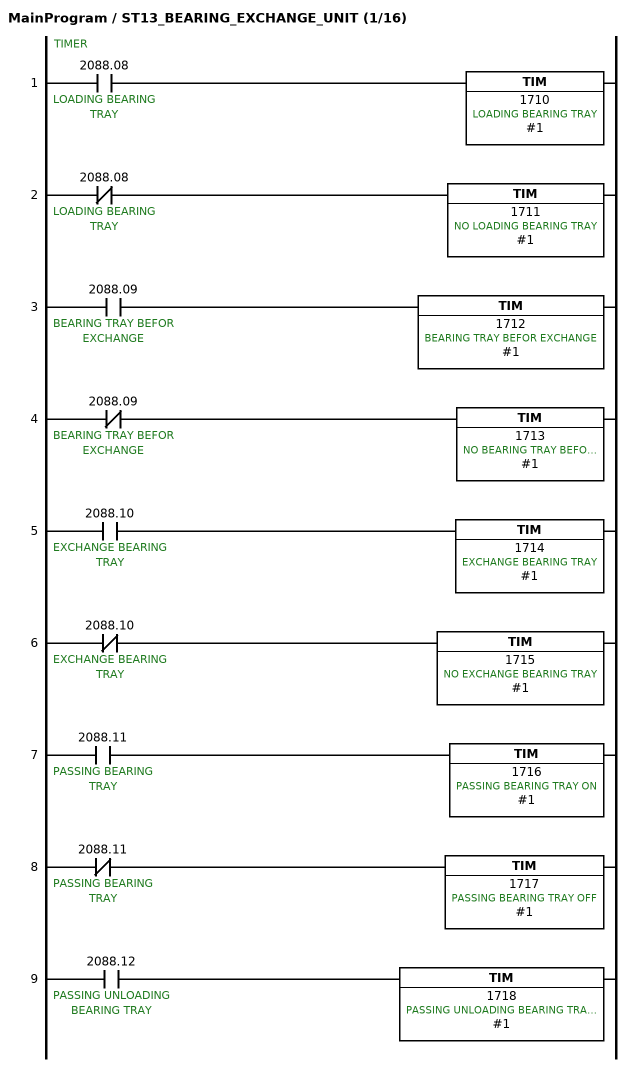
; rung 1: TIMER
LD 2088.08  ; LOADING BEARING TRAY
TIM 1710 #1  ; LOADING BEARING TRAY
; rung 2
LDNOT 2088.08  ; LOADING BEARING TRAY
TIM 1711 #1  ; NO LOADING BEARING TRAY
; rung 3
LD 2088.09  ; BEARING TRAY BEFOR EXCHANGE
TIM 1712 #1  ; BEARING TRAY BEFOR EXCHANGE
; rung 4
LDNOT 2088.09  ; BEARING TRAY BEFOR EXCHANGE
TIM 1713 #1  ; NO BEARING TRAY BEFOR EXCHANGE
; rung 5
LD 2088.10  ; EXCHANGE BEARING TRAY
TIM 1714 #1  ; EXCHANGE BEARING TRAY
; rung 6
LDNOT 2088.10  ; EXCHANGE BEARING TRAY
TIM 1715 #1  ; NO EXCHANGE BEARING TRAY
; rung 7
LD 2088.11  ; PASSING BEARING TRAY
TIM 1716 #1  ; PASSING BEARING TRAY ON
; rung 8
LDNOT 2088.11  ; PASSING BEARING TRAY
TIM 1717 #1  ; PASSING BEARING TRAY OFF
; rung 9
LD 2088.12  ; PASSING UNLOADING BEARING TRAY
TIM 1718 #1  ; PASSING UNLOADING BEARING TRAY ON

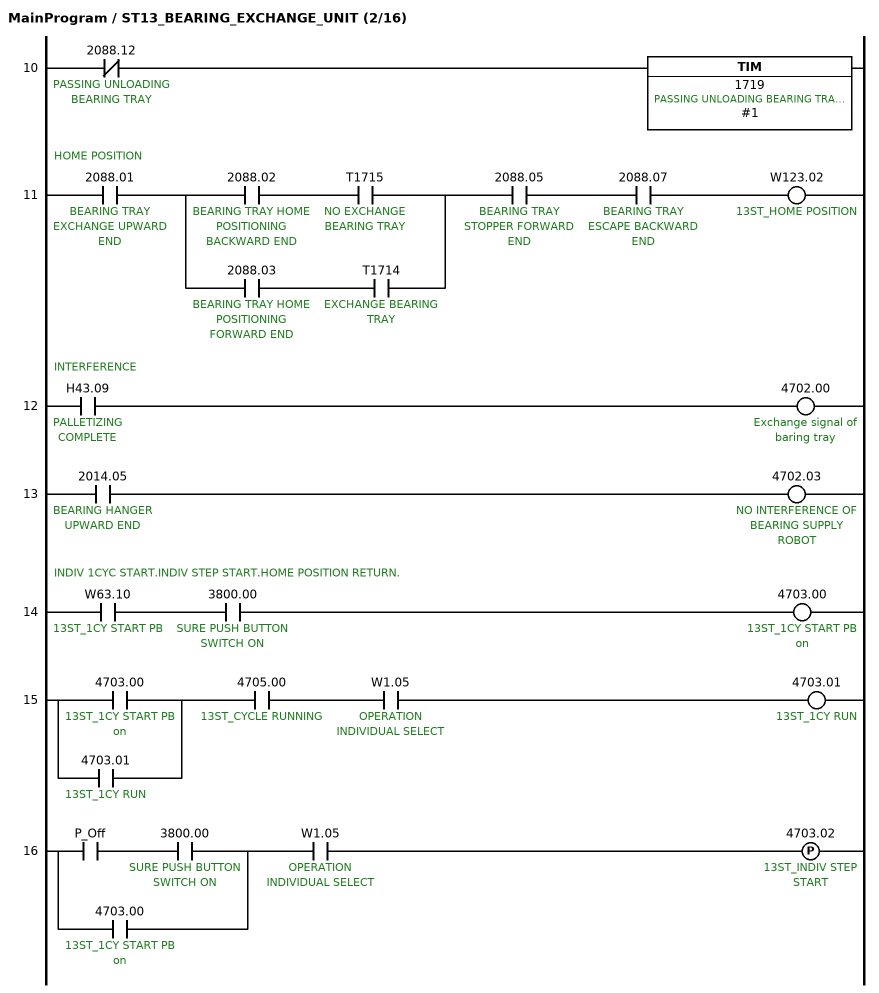
; rung 10
LDNOT 2088.12  ; PASSING UNLOADING BEARING TRAY
TIM 1719 #1  ; PASSING UNLOADING BEARING TRAY OFF
; rung 11: HOME POSITION
LD 2088.01  ; BEARING TRAY EXCHANGE UPWARD END
LD 2088.02  ; BEARING TRAY HOME POSITIONING BACKWARD END
AND T1715  ; NO EXCHANGE BEARING TRAY
LD 2088.03  ; BEARING TRAY HOME POSITIONING FORWARD END
AND T1714  ; EXCHANGE BEARING TRAY
ORLD
ANDLD
AND 2088.05  ; BEARING TRAY STOPPER FORWARD END
AND 2088.07  ; BEARING TRAY ESCAPE BACKWARD END
OUT W123.02  ; 13ST_HOME POSITION
; rung 12: INTERFERENCE
LD H43.09  ; PALLETIZING COMPLETE
OUT 4702.00  ; Exchange signal of baring tray
; rung 13
LD 2014.05  ; BEARING HANGER UPWARD END
OUT 4702.03  ; NO INTERFERENCE OF BEARING SUPPLY ROBOT
; rung 14: INDIV 1CYC START.INDIV STEP START.HOME POSITION RETURN.
LD W63.10  ; 13ST_1CY START PB
AND 3800.00  ; SURE PUSH BUTTON SWITCH ON
OUT 4703.00  ; 13ST_1CY START PB on
; rung 15
LD 4703.00  ; 13ST_1CY START PB on
OR 4703.01  ; 13ST_1CY RUN
AND 4705.00  ; 13ST_CYCLE RUNNING
AND W1.05  ; OPERATION INDIVIDUAL SELECT
OUT 4703.01  ; 13ST_1CY RUN
; rung 16
LD P_Off
AND 3800.00  ; SURE PUSH BUTTON SWITCH ON
OR 4703.00  ; 13ST_1CY START PB on
AND W1.05  ; OPERATION INDIVIDUAL SELECT
DIFU(013) 4703.02  ; 13ST_INDIV STEP START

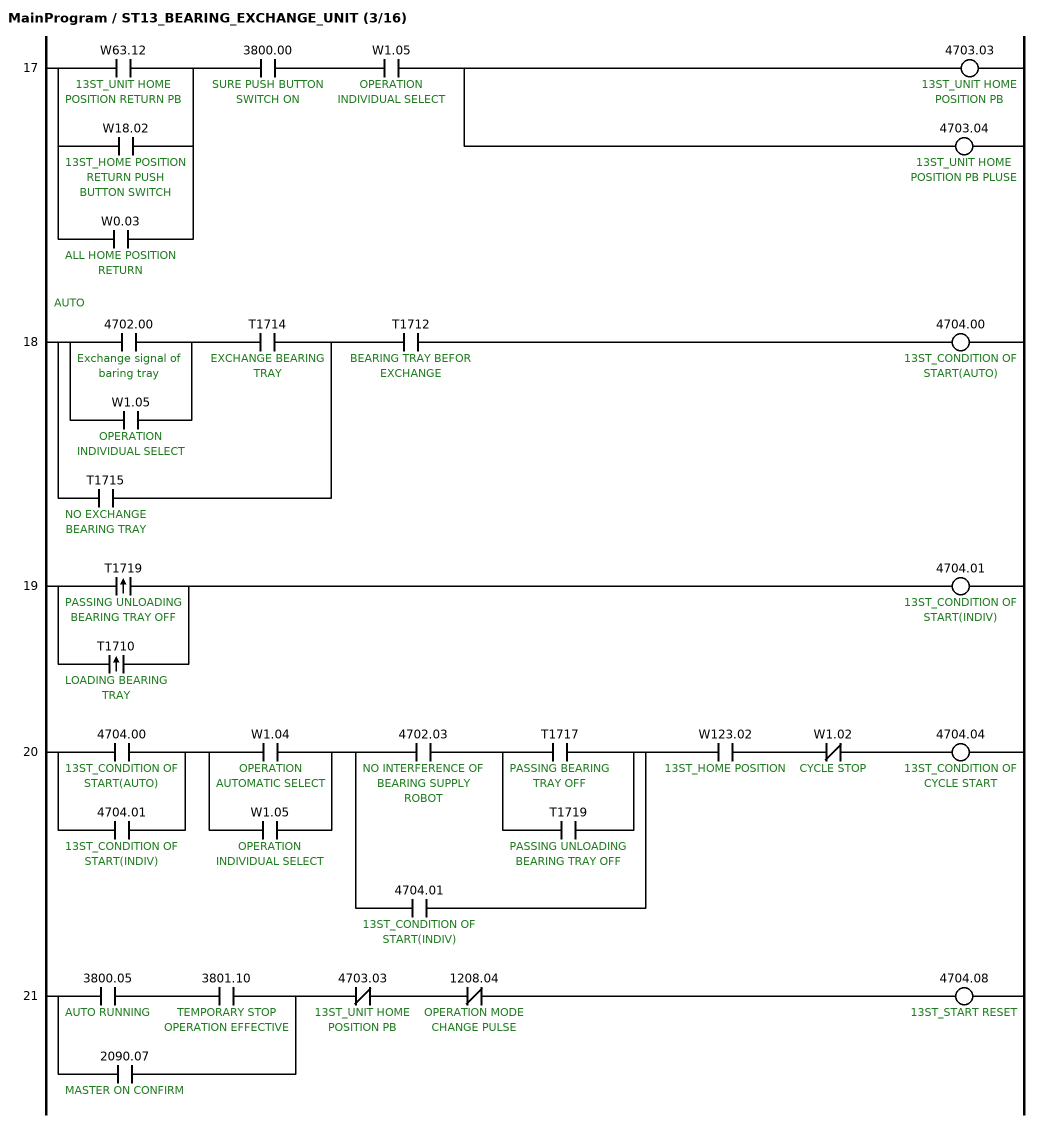
; rung 17
LD W63.12  ; 13ST_UNIT HOME POSITION RETURN PB
OR W18.02  ; 13ST_HOME POSITION RETURN PUSH BUTTON SWITCH
OR W0.03  ; ALL HOME POSITION RETURN
AND 3800.00  ; SURE PUSH BUTTON SWITCH ON
AND W1.05  ; OPERATION INDIVIDUAL SELECT
OUT 4703.03  ; 13ST_UNIT HOME POSITION PB
OUT 4703.04  ; 13ST_UNIT HOME POSITION PB PLUSE
; rung 18: AUTO
LD 4702.00  ; Exchange signal of baring tray
OR W1.05  ; OPERATION INDIVIDUAL SELECT
AND T1714  ; EXCHANGE BEARING TRAY
OR T1715  ; NO EXCHANGE BEARING TRAY
AND T1712  ; BEARING TRAY BEFOR EXCHANGE
OUT 4704.00  ; 13ST_CONDITION OF START(AUTO)
; rung 19
@LD T1719  ; PASSING UNLOADING BEARING TRAY OFF
@OR T1710  ; LOADING BEARING TRAY
OUT 4704.01  ; 13ST_CONDITION OF START(INDIV)
; rung 20
LD 4704.00  ; 13ST_CONDITION OF START(AUTO)
OR 4704.01  ; 13ST_CONDITION OF START(INDIV)
LD W1.04  ; OPERATION AUTOMATIC SELECT
OR W1.05  ; OPERATION INDIVIDUAL SELECT
ANDLD
LD 4702.03  ; NO INTERFERENCE OF BEARING SUPPLY ROBOT
LD T1717  ; PASSING BEARING TRAY OFF
OR T1719  ; PASSING UNLOADING BEARING TRAY OFF
ANDLD
OR 4704.01  ; 13ST_CONDITION OF START(INDIV)
ANDLD
AND W123.02  ; 13ST_HOME POSITION
ANDNOT W1.02  ; CYCLE STOP
OUT 4704.04  ; 13ST_CONDITION OF CYCLE START
; rung 21
LD 3800.05  ; AUTO RUNNING
AND 3801.10  ; TEMPORARY STOP OPERATION EFFECTIVE
OR 2090.07  ; MASTER ON CONFIRM
ANDNOT 4703.03  ; 13ST_UNIT HOME POSITION PB
ANDNOT 1208.04  ; OPERATION MODE CHANGE PULSE
OUT 4704.08  ; 13ST_START RESET

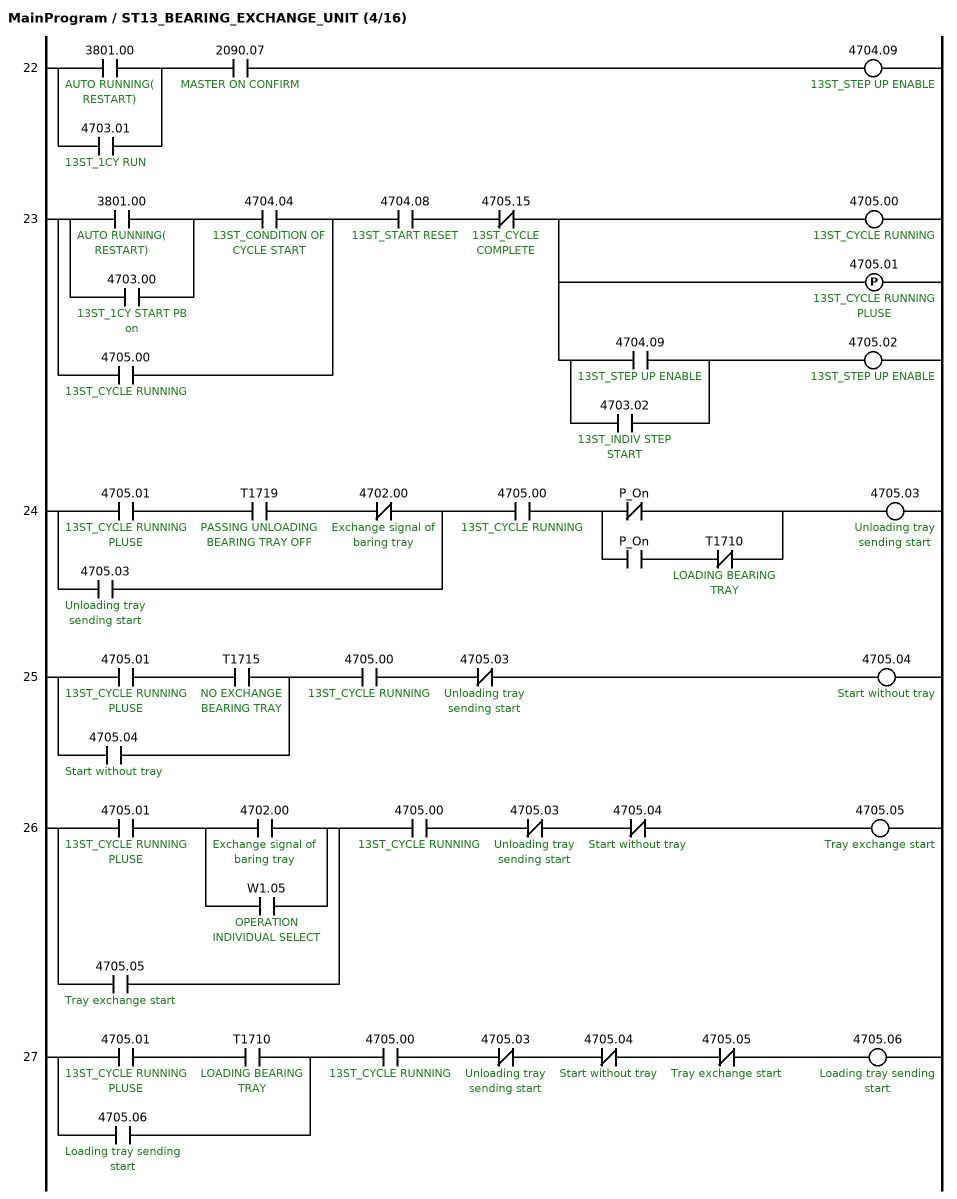
; rung 22
LD 3801.00  ; AUTO RUNNING(RESTART)
OR 4703.01  ; 13ST_1CY RUN
AND 2090.07  ; MASTER ON CONFIRM
OUT 4704.09  ; 13ST_STEP UP ENABLE
; rung 23
LD 3801.00  ; AUTO RUNNING(RESTART)
OR 4703.00  ; 13ST_1CY START PB on
AND 4704.04  ; 13ST_CONDITION OF CYCLE START
OR 4705.00  ; 13ST_CYCLE RUNNING
AND 4704.08  ; 13ST_START RESET
ANDNOT 4705.15  ; 13ST_CYCLE COMPLETE
OUT 4705.00  ; 13ST_CYCLE RUNNING
DIFU(013) 4705.01  ; 13ST_CYCLE RUNNING PLUSE
LD 4704.09  ; 13ST_STEP UP ENABLE
OR 4703.02  ; 13ST_INDIV STEP START
ANDLD
OUT 4705.02  ; 13ST_STEP UP ENABLE
; rung 24
LD 4705.01  ; 13ST_CYCLE RUNNING PLUSE
AND T1719  ; PASSING UNLOADING BEARING TRAY OFF
ANDNOT 4702.00  ; Exchange signal of baring tray
OR 4705.03  ; Unloading tray sending start
AND 4705.00  ; 13ST_CYCLE RUNNING
LDNOT P_On
LD P_On
ANDNOT T1710  ; LOADING BEARING TRAY
ORLD
ANDLD
OUT 4705.03  ; Unloading tray sending start
; rung 25
LD 4705.01  ; 13ST_CYCLE RUNNING PLUSE
AND T1715  ; NO EXCHANGE BEARING TRAY
OR 4705.04  ; Start without tray
AND 4705.00  ; 13ST_CYCLE RUNNING
ANDNOT 4705.03  ; Unloading tray sending start
OUT 4705.04  ; Start without tray
; rung 26
LD 4705.01  ; 13ST_CYCLE RUNNING PLUSE
LD 4702.00  ; Exchange signal of baring tray
OR W1.05  ; OPERATION INDIVIDUAL SELECT
ANDLD
OR 4705.05  ; Tray exchange start
AND 4705.00  ; 13ST_CYCLE RUNNING
ANDNOT 4705.03  ; Unloading tray sending start
ANDNOT 4705.04  ; Start without tray
OUT 4705.05  ; Tray exchange start
; rung 27
LD 4705.01  ; 13ST_CYCLE RUNNING PLUSE
AND T1710  ; LOADING BEARING TRAY
OR 4705.06  ; Loading tray sending start
AND 4705.00  ; 13ST_CYCLE RUNNING
ANDNOT 4705.03  ; Unloading tray sending start
ANDNOT 4705.04  ; Start without tray
ANDNOT 4705.05  ; Tray exchange start
OUT 4705.06  ; Loading tray sending start

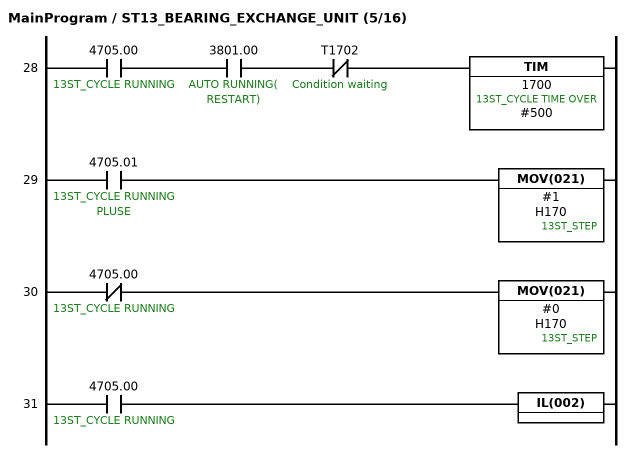
; rung 28
LD 4705.00  ; 13ST_CYCLE RUNNING
AND 3801.00  ; AUTO RUNNING(RESTART)
ANDNOT T1702  ; Condition waiting
TIM 1700 #500  ; 13ST_CYCLE TIME OVER
; rung 29
LD 4705.01  ; 13ST_CYCLE RUNNING PLUSE
MOV(021) #1 H170  ; 13ST_STEP
; rung 30
LDNOT 4705.00  ; 13ST_CYCLE RUNNING
MOV(021) #0 H170  ; 13ST_STEP
; rung 31
LD 4705.00  ; 13ST_CYCLE RUNNING
IL(002)

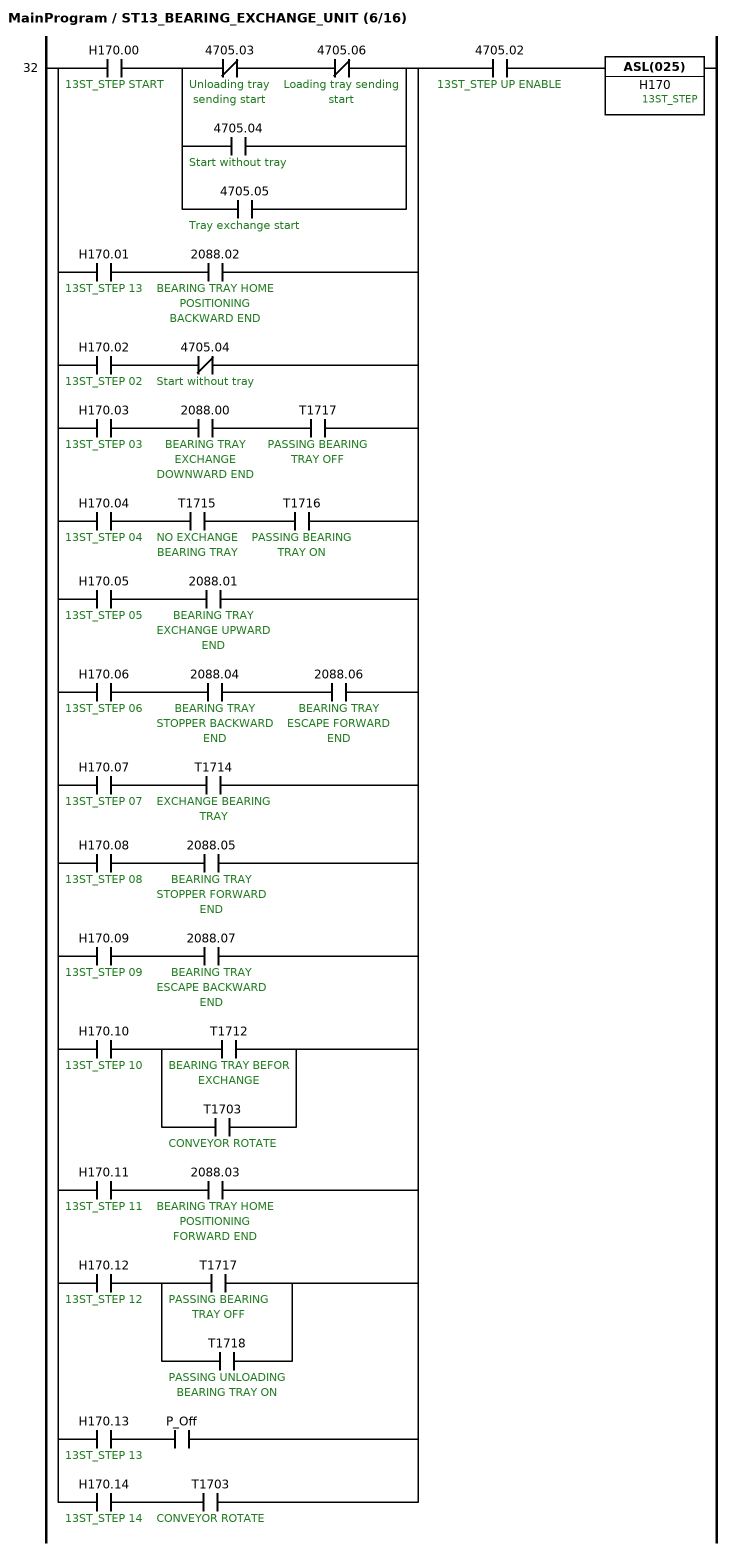
; rung 32
LD H170.00  ; 13ST_STEP START
LDNOT 4705.03  ; Unloading tray sending start
ANDNOT 4705.06  ; Loading tray sending start
OR 4705.04  ; Start without tray
OR 4705.05  ; Tray exchange start
ANDLD
LD H170.01  ; 13ST_STEP 13
AND 2088.02  ; BEARING TRAY HOME POSITIONING BACKWARD END
ORLD
LD H170.02  ; 13ST_STEP 02
ANDNOT 4705.04  ; Start without tray
ORLD
LD H170.03  ; 13ST_STEP 03
AND 2088.00  ; BEARING TRAY EXCHANGE DOWNWARD END
AND T1717  ; PASSING BEARING TRAY OFF
ORLD
LD H170.04  ; 13ST_STEP 04
AND T1715  ; NO EXCHANGE BEARING TRAY
AND T1716  ; PASSING BEARING TRAY ON
ORLD
LD H170.05  ; 13ST_STEP 05
AND 2088.01  ; BEARING TRAY EXCHANGE UPWARD END
ORLD
LD H170.06  ; 13ST_STEP 06
AND 2088.04  ; BEARING TRAY STOPPER BACKWARD END
AND 2088.06  ; BEARING TRAY ESCAPE FORWARD END
ORLD
LD H170.07  ; 13ST_STEP 07
AND T1714  ; EXCHANGE BEARING TRAY
ORLD
LD H170.08  ; 13ST_STEP 08
AND 2088.05  ; BEARING TRAY STOPPER FORWARD END
ORLD
LD H170.09  ; 13ST_STEP 09
AND 2088.07  ; BEARING TRAY ESCAPE BACKWARD END
ORLD
LD H170.10  ; 13ST_STEP 10
LD T1712  ; BEARING TRAY BEFOR EXCHANGE
OR T1703  ; CONVEYOR ROTATE
ANDLD
ORLD
LD H170.11  ; 13ST_STEP 11
AND 2088.03  ; BEARING TRAY HOME POSITIONING FORWARD END
ORLD
LD H170.12  ; 13ST_STEP 12
LD T1717  ; PASSING BEARING TRAY OFF
OR T1718  ; PASSING UNLOADING BEARING TRAY ON
ANDLD
ORLD
LD H170.13  ; 13ST_STEP 13
AND P_Off
ORLD
LD H170.14  ; 13ST_STEP 14
AND T1703  ; CONVEYOR ROTATE
ORLD
AND 4705.02  ; 13ST_STEP UP ENABLE
ASL(025) H170  ; 13ST_STEP

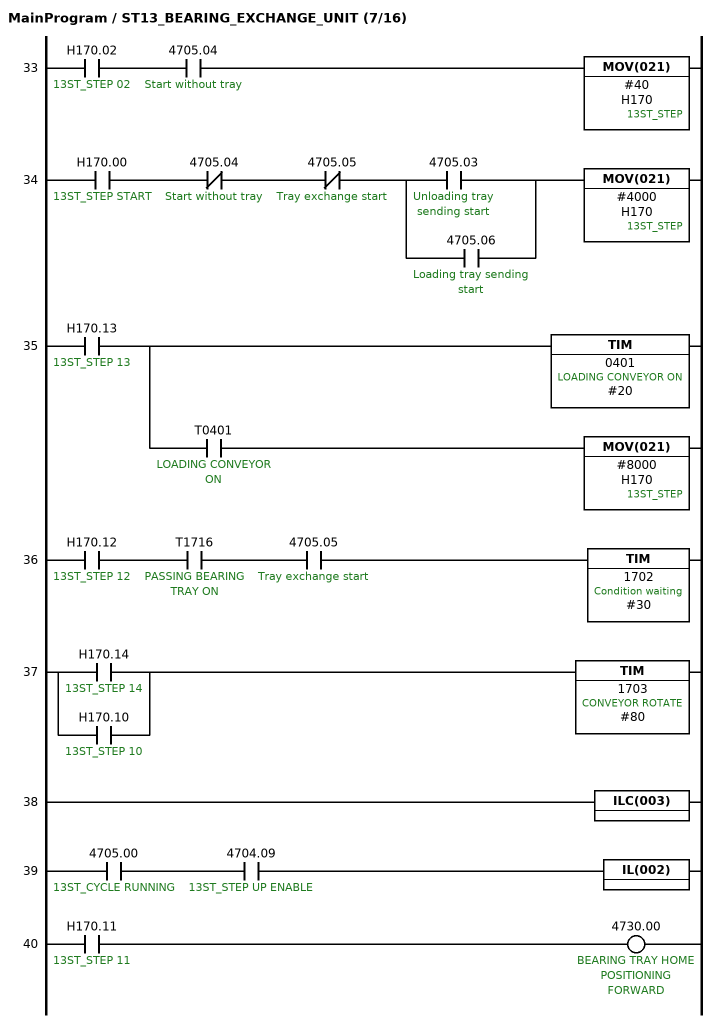
; rung 33
LD H170.02  ; 13ST_STEP 02
AND 4705.04  ; Start without tray
MOV(021) #40 H170  ; 13ST_STEP
; rung 34
LD H170.00  ; 13ST_STEP START
ANDNOT 4705.04  ; Start without tray
ANDNOT 4705.05  ; Tray exchange start
LD 4705.03  ; Unloading tray sending start
OR 4705.06  ; Loading tray sending start
ANDLD
MOV(021) #4000 H170  ; 13ST_STEP
; rung 35
LD H170.13  ; 13ST_STEP 13
TIM 0401 #20  ; LOADING CONVEYOR ON
AND T0401  ; LOADING CONVEYOR ON
MOV(021) #8000 H170  ; 13ST_STEP
; rung 36
LD H170.12  ; 13ST_STEP 12
AND T1716  ; PASSING BEARING TRAY ON
AND 4705.05  ; Tray exchange start
TIM 1702 #30  ; Condition waiting
; rung 37
LD H170.14  ; 13ST_STEP 14
OR H170.10  ; 13ST_STEP 10
TIM 1703 #80  ; CONVEYOR ROTATE
; rung 38
ILC(003)
; rung 39
LD 4705.00  ; 13ST_CYCLE RUNNING
AND 4704.09  ; 13ST_STEP UP ENABLE
IL(002)
; rung 40
LD H170.11  ; 13ST_STEP 11
OUT 4730.00  ; BEARING TRAY HOME POSITIONING FORWARD

